// TIA Portal V20 export
FUNCTION_BLOCK "FB_TimeMeasure"   // FB51, SCL
{ S7_Optimized_Access := 'TRUE' }
// stored: AutoNumber false, MemoryReserve 100, SetENOAutomatically false
   VAR_INPUT
      iImpulsion : Bool;
      iPLC_DateAndTime : DTL;
   END_VAR
   VAR
      sRT_Impuls : R_TRIG;
      sRT_Impuls1 : R_TRIG;
      sRT_Impuls2 { S7_SetPoint := 'True'} : R_TRIG;
      sTime1 { S7_SetPoint := 'True'} : DTL;
      sTime2 : DTL;
      sDeltaTime : LTime;
      sToggleStatus : Bool;
   END_VAR
BEGIN
   REGION Description header 
       //==================================================================================
       // POSALUX Swiss SA / (C) Copyright 2026
       //----------------------------------------------------------------------------------
       // Title: FB_TimeMeasure
       // Comment/Function: This function allows:
       //                      - Counting Time between 2 pulses
       //
       // Author: Fabien Waldt
       // Engineering: TIA Portal v20
       //----------------------------------------------------------------------------------
       // Change log table:
       // Version  | Date     | Expert in charge | Changes applied
       // ---------|----------|------------------|------------------------------------
       // 00.00.01 | 20261211 | WFA              | First released version
       // ==================================================================================
   END_REGION

   REGION Delta time calculation
       // Rising edge detection
       #sRT_Impuls(CLK := #iImpulsion);

       // Toggle state update
       IF #sRT_Impuls.Q THEN
           #sToggleStatus := NOT #sToggleStatus;
       END_IF;
       #sRT_Impuls1(CLK := #sToggleStatus);
       #sRT_Impuls2(CLK := NOT #sToggleStatus);

       // Timestamp of the first rising edge
       IF #sRT_Impuls1.Q THEN
           #sTime1 := #iPLC_DateAndTime;
       END_IF;

       // Timestamp of the second rising edge + calculation
       IF #sRT_Impuls2.Q THEN
           #sTime2 := #iPLC_DateAndTime;
           #sDeltaTime := #sTime2 - #sTime1;
       END_IF;
   END_REGION
END_FUNCTION_BLOCK
